// TIA Portal V18 export
TYPE "UDT_Vitotronic100_IOs"
// stored: IsFailsafeCompliant false
   STRUCT
      "Boiler water temperature" : Array[0..2] of Real;
      "Flue gas temperature" : Array[0..2] of Real;
      "Return temperature 17A" : Array[0..2] of Real;
      "Return temperature 17B" : Array[0..2] of Real;
   END_STRUCT;
END_TYPE
